// Mitsubishi GX Works2 project: StBlock1   PLC: Q03UDV

// task Task_01 (event TRUE, interval 0, priority 31): POU_01
// task stBlock (event TRUE, interval 0, priority 31): stBlock

PROGRAM POU_01
VAR
  CTD_1 : CTD;
  counter1 : BOOL;
  CTU_1 : CTU;
  counter2 : BOOL;
  CTU_2 : CTU;
  TP_1 : TP;
  TIMER1 : BOOL;
  TON_1 : TON;
  TIMER2 : BOOL;
  TOF_1 : TOF;
  TOF_2 : TOF;
  TIMER3 : BOOL;
  TimerTP : TIME;
  TimeON : TIME;
  TimeOFF : TIME;
END_VAR
(* structured ladder/FBD written out as ST: instructions are called as NAME(EN, inputs, outputs); _pN, _eN, _tN stand for wires *)
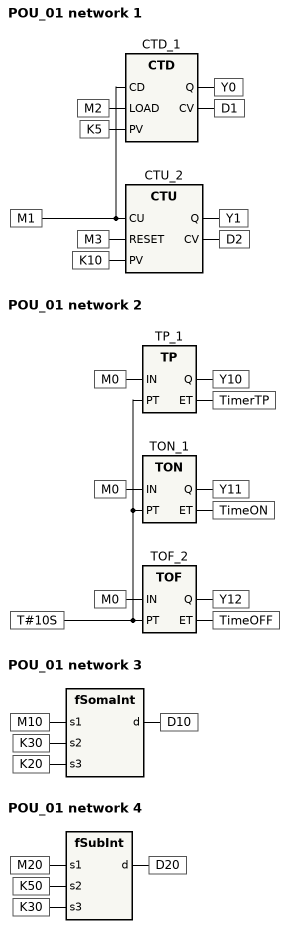
(* network 1 *)
CTD_1(CD := M1, LOAD := M2, PV := K5, Q => Y0, CV => D1);
CTU_2(CU := M1, RESET := M3, PV := K10, Q => Y1, CV => D2);
(* network 2 *)
TP_1(IN := M0, PT := T#10S, Q => Y10, ET => TimerTP);
TON_1(IN := M0, PT := T#10S, Q => Y11, ET => TimeON);
TOF_2(IN := M0, PT := T#10S, Q => Y12, ET => TimeOFF);
(* network 3 *)
D10 := fSomaInt(M10, K30, K20);
(* network 4 *)
D20 := fSubInt(M20, K50, K30);
END_PROGRAM

FUNCTION fSomaInt
VAR_INPUT
  i_xHabilitar : BOOL;
  i_iElemento1 : INT;
  i_iElemento2 : INT;
END_VAR
(* structured ladder/FBD written out as ST: instructions are called as NAME(EN, inputs, outputs); _pN, _eN, _tN stand for wires *)
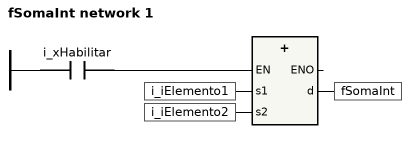
(* network 1 *)
+(i_xHabilitar, i_iElemento1, i_iElemento2, fSomaInt);
END_FUNCTION

FUNCTION fSubInt
VAR_INPUT
  i_xHabilita2 : BOOL;
  i_iElemento2 : INT;
  i_iElemento3 : INT;
END_VAR
(* structured ladder/FBD written out as ST: instructions are called as NAME(EN, inputs, outputs); _pN, _eN, _tN stand for wires *)
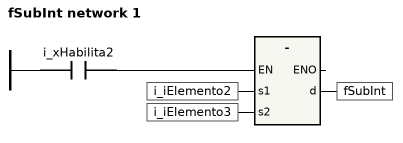
(* network 1 *)
-(i_xHabilita2, i_iElemento2, i_iElemento3, fSubInt);
END_FUNCTION

FUNCTION fMulInt
VAR_INPUT
  i_xHabilita3 : BOOL;
  i_iElemento5 : INT;
  i_iElemento4 : INT;
END_VAR
(* structured ladder/FBD written out as ST: instructions are called as NAME(EN, inputs, outputs); _pN, _eN, _tN stand for wires *)
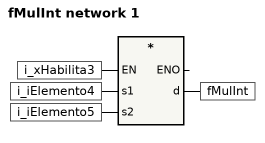
(* network 1 *)
*(i_xHabilita3, i_iElemento4, i_iElemento5, fMulInt);
END_FUNCTION

PROGRAM stBlock
VAR CONSTANT
  iEle01 : INT := 15;
  iEle02 : INT := 4;
END_VAR
VAR
  iDR : ARRAY [0..4] OF INT;
  xEnable : BOOL;
  iDR1 : ARRAY [0..1] OF INT;
  iDR2 : ARRAY [0..1] OF DINT;
  xEnableOperation : BOOL;
  Result : INT;
  i_xHabilitar5 : BOOL;
  i_iValor1 : INT;
  i_iValor2 : INT;
  OperadorMat : STRING[32];
  Result1 : INT;
END_VAR
iDR[0]:=iEle01+iEle02;
iDR[1]:=iEle01-iEle02;
iDR[2]:=iEle01*iEle02;
iDR[3]:=iEle01/iEle02;
iDR[4]:= iEle01 MOD iEle02;

iDR1[0]:= fSomaInt( xEnable , iEle01 , iEle02 );
iDR1[1]:= fSubInt( xEnable, iEle01 , iEle02 );
iDR2[0]:= fMulInt( xEnable, iEle01, iEle02 );
(*iDR2[1]:= fDivInt( xEnable , iEle01, iEle02 );*)

IF xEnableOperation THEN
	iDR[0]:= iEle01 + iEle02;
ELSE
	iDR[0]:= iEle01 - iEle02;
END_IF;

Result := fCondicionalIf( i_xHabilitar5 , i_iValor1 , i_iValor2, OperadorMat );
END_PROGRAM

FUNCTION fDivInt
VAR_INPUT
  i_xHabilita4 : BOOL;
  i_iElemento6 : INT;
  i_iElemento7 : INT;
END_VAR
(* structured ladder/FBD written out as ST: instructions are called as NAME(EN, inputs, outputs); _pN, _eN, _tN stand for wires *)
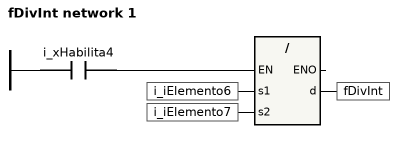
(* network 1 *)
/(i_xHabilita4, i_iElemento6, i_iElemento7, fDivInt);
END_FUNCTION

FUNCTION fCondicionalIf
VAR_INPUT
  i_iValor1 : INT;
  i_iValor2 : INT;
  OperadorMat : STRING[32];
  i_xHabilitar5 : BOOL;
END_VAR
IF i_xHabilitar5 THEN
	IF OperadorMat="+" THEN
		fCondicionalIf:= i_iValor1+i_iValor2;
	ELSIF
		OperadorMat="-" THEN
		fCondicionalIf:= i_iValor1-i_iValor2;
	ELSIF
		OperadorMat="*" THEN
		fCondicionalIf:= i_iValor1*i_iValor2;
	ELSIF
		OperadorMat = "/" THEN
		fCondicionalIf:= i_iValor1/i_iValor2;
	ELSIF
		(OperadorMat= "Mod") OR (OperadorMat = "M") THEN
		fCondicionalIf:= i_iValor1 MOD i_iValor2;
	ELSE
		fCondicionalIf:= 32767;
	END_IF;
	ELSE
	fCondicionalIf:= -32767;
END_IF;
END_FUNCTION
